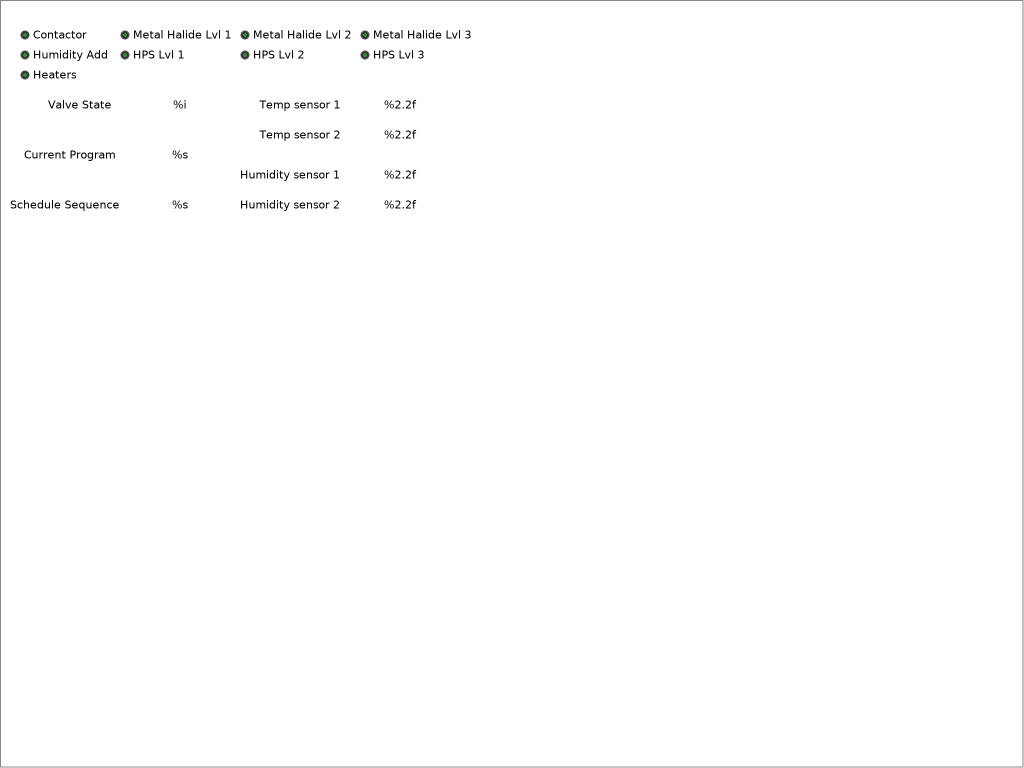
VISUALIZATION IO  // 1024x768
    Lamp1 (20,30 10x10), variable: IO_VARS.ENABLE, style: Lamp-Lamp1-Green
    Label (30,20 100x30), "Contactor"
    Textfield (130,140 100x30), "%s", text variable: GVL.CurrentProgramName
    Label (20,140 100x30), "Current Program"
    Label (10,190 110x30), "Schedule Sequence"
    Textfield (130,190 100x30), "%s", text variable: GVL.ScheduleSequence
    Textfield (130,90 100x30), "%i", text variable: GVL.iTempControl
    Label (30,90 100x30), "Valve State"
    Lamp1 (120,30 10x10), variable: IO_VARS.FL1, style: Lamp-Lamp1-Green
    Label (130,20 100x30), "Metal Halide Lvl 1"
    Lamp1 (240,30 10x10), variable: IO_VARS.FL2, style: Lamp-Lamp1-Green
    Label (250,20 100x30), "Metal Halide Lvl 2"
    Lamp1 (360,30 10x10), variable: IO_VARS.FL3, style: Lamp-Lamp1-Green
    Label (370,20 100x30), "Metal Halide Lvl 3"
    Lamp1 (120,50 10x10), variable: IO_VARS.HPS1, style: Lamp-Lamp1-Green
    Label (130,40 100x30), "HPS Lvl 1"
    Lamp1 (240,50 10x10), variable: IO_VARS.HPS2, style: Lamp-Lamp1-Green
    Label (250,40 100x30), "HPS Lvl 2"
    Lamp1 (360,50 10x10), variable: IO_VARS.HPS3, style: Lamp-Lamp1-Green
    Label (370,40 100x30), "HPS Lvl 3"
    Label (30,40 100x30), "Humidity Add"
    Lamp1 (20,50 10x10), variable: IO_VARS.HUMVALVE, style: Lamp-Lamp1-Green
    Label (30,60 100x30), "Heaters"
    Lamp1 (20,70 10x10), variable: IO_VARS.HEATERS, style: Lamp-Lamp1-Green
    Label (250,90 100x30), "Temp sensor 1"
    Textfield (350,90 100x30), "%2.2f", text variable: GVL.Temp
    Label (250,120 100x30), "Temp sensor 2"
    Textfield (350,120 100x30), "%2.2f", text variable: GVL.Temp2
    Label (230,160 120x30), "Humidity sensor 1"
    Textfield (350,160 100x30), "%2.2f", text variable: GVL.Humidity
    Label (230,190 120x30), "Humidity sensor 2"
    Textfield (350,190 100x30), "%2.2f", text variable: GVL.Humidity2
END_VISUALIZATION

(* stored: Version 1.1.0.1, ProductVersion 3.1.4022.18
   Visu IO: Id {92aa4d61-b6ee-4756-badc-04c62c80f55c} *)
